Staubli VAL3: getPoint.pgx

public program getPoint(point& x_pPoint[], bool x_bCycle, num x_nIndex)
  local string l_sItem
  local tool l_tTool
begin
  // take
  // check the point
  link(x_pPoint,world)
  if x_bCycle
    call tcp:getTool(l_tTool,pt:tTraj[sTrajCycle].nIndexTool)
    x_pPoint=jointToPoint(l_tTool,world,pt:tTraj[sTrajCycle].tData[x_nIndex].jJoint)
  else
    // give back the point
    call tcp:getTool(l_tTool,jEditPoint.nIndexTool)
    x_pPoint=jointToPoint(l_tTool,world,jEditPoint.tData[x_nIndex].jJoint)
  endIf
end
